INTERFACE I_SessionData EXTENDS I_Disposable

END_INTERFACE

(* stored: Version 1.1.0.1, ProductVersion 3.1.4026.13
   Itf I_SessionData: Id {412509da-d3de-460f-a3e6-bed4ca3b46f8} *)
